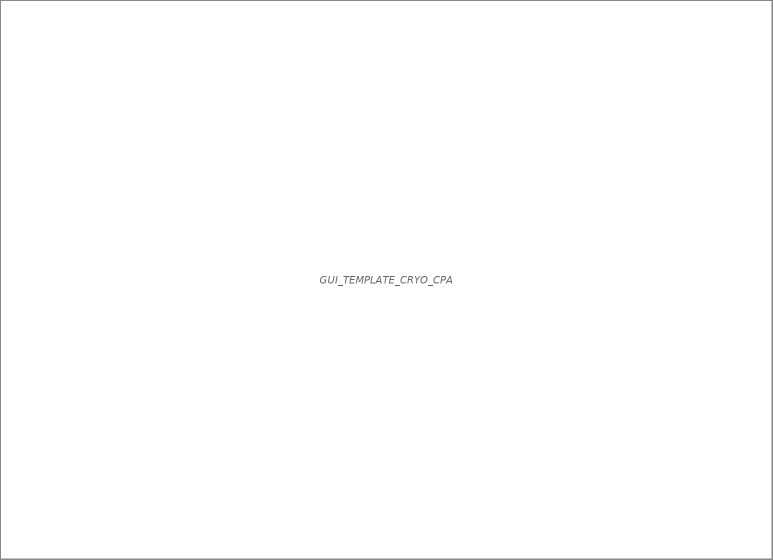
VISUALIZATION GUI_CPA  // 773x560
    Frame (0,0 773x560)
        shows GUI_TEMPLATE_CRYO_CPA(m_Instance := MAIN.Cryo_Ctrl.cpa)
END_VISUALIZATION

(* stored: Version 1.1.0.1, ProductVersion 3.1.4024.9
   Visu GUI_CPA: Id {536f4479-67b8-4c28-94d4-83c3196e8779} *)
